Fanuc KAREL source: kb00011.KL

-- PROVISIONAL review KL for V770-1; original PC SHA256 1b2729f573180ed3cb5cc168b820d21e9e49324e56a3c63e368d849e140c7c59
-- Incomplete behavior may be omitted. Consult companion uncertainty JSON. Do not deploy.
PROGRAM KB00011
%NOLOCKGROUP
BEGIN
  -- UNRESOLVED_PC offsets 5-14; opcodes 3F,75
  -- UNRESOLVED_PC offsets 19-28; opcodes 3F,75
  -- UNRESOLVED_PC offsets 33-40; opcodes 9D,23
  -- UNRESOLVED_PC offsets 45-52; opcodes 9D,23
  -- UNRESOLVED_PC offsets 57-64; opcodes 9D,23
  -- UNRESOLVED_PC offsets 69-107; opcodes 27,22,2A,22,2A,22,22,22,31
  -- UNRESOLVED_PC offsets 112-116; opcodes 7F
END KB00011
